# EPICS autosave request: bcurApp/Db/pipette_settings.req
$(P)Pipette:SetPlunger.VAL
$(P)Pipette:SetSpeed.VAL
$(P)Pipette:SetDeadVolume.VAL
$(P)Pipette:SetVolume.VAL
